# EPICS alarm handler configuration: mps_database/bare/alarms/areas/mpln_dog_mp05.alhConfig
GROUP NULL MPLN:DOG:MP05:1
$ALIAS MPS Link Node 76
$GUIDANCE
LTUH MPS
   Group Name: MPLN:DOG:MP05:1
   Summary PV:  MPLN:DOG:MP05:1:STATSUMY
$END
CHANNEL  MPLN:DOG:MP05:1    MPLN:DOG:MP05:1:MPS_EN_RBV		-----
CHANNEL  MPLN:DOG:MP05:1    MPLN:DOG:MP05:1:LC1_MODE_RBV		-----
